GLOBALCONSTANTS DefaultPool_Numeric (* Numeric object pool constants (ID, Scale, Offset, Decimals) *)
  PACKAGE test::FBs::Baumsetzer::Constants;
  VAR_GLOBAL CONSTANT
    InputNumber_Pflanzabstand : logiBUS::utils::conversion::phys::NumericObjectPool_S := (u16ObjId := 9001, r32Scale := 0.001, i32Offset := 0, u8Decimals := 3);
    InputNumber_Luftversatz : logiBUS::utils::conversion::phys::NumericObjectPool_S := (u16ObjId := 9002, r32Scale := 0.1, i32Offset := 0, u8Decimals := 1);
    InputNumber_Wasserversatz : logiBUS::utils::conversion::phys::NumericObjectPool_S := (u16ObjId := 9003, r32Scale := 0.1, i32Offset := 0, u8Decimals := 1);
    InputNumber_Granulatversatz : logiBUS::utils::conversion::phys::NumericObjectPool_S := (u16ObjId := 9004, r32Scale := 0.1, i32Offset := 0, u8Decimals := 1);
    InputNumber_Summer_Dauer : logiBUS::utils::conversion::phys::NumericObjectPool_S := (u16ObjId := 9005, r32Scale := 1.0, i32Offset := 0, u8Decimals := 0);
    InputNumber_Luft_Dauer : logiBUS::utils::conversion::phys::NumericObjectPool_S := (u16ObjId := 9006, r32Scale := 1.0, i32Offset := 0, u8Decimals := 0);
    InputNumber_Wasser_Dauer : logiBUS::utils::conversion::phys::NumericObjectPool_S := (u16ObjId := 9007, r32Scale := 1.0, i32Offset := 0, u8Decimals := 0);
    InputNumber_Granulat_Dauer : logiBUS::utils::conversion::phys::NumericObjectPool_S := (u16ObjId := 9008, r32Scale := 1.0, i32Offset := 0, u8Decimals := 0);
    OutputNumber_12000 : logiBUS::utils::conversion::phys::NumericObjectPool_S := (u16ObjId := 12000, r32Scale := 0.0036, i32Offset := 0, u8Decimals := 1);
    Einsatzstunden : logiBUS::utils::conversion::phys::NumericObjectPool_S := (u16ObjId := 12001, r32Scale := 1.0, i32Offset := 0, u8Decimals := 0);
    Einsatzminuten : logiBUS::utils::conversion::phys::NumericObjectPool_S := (u16ObjId := 12002, r32Scale := 1.0, i32Offset := 0, u8Decimals := 0);
    OutputNumber_Baeume_gepflanzt : logiBUS::utils::conversion::phys::NumericObjectPool_S := (u16ObjId := 12003, r32Scale := 1.0, i32Offset := 0, u8Decimals := 0);
    OutputNumber_12004 : logiBUS::utils::conversion::phys::NumericObjectPool_S := (u16ObjId := 12004, r32Scale := 0.0036, i32Offset := 0, u8Decimals := 1);
    OutputNumber_12005 : logiBUS::utils::conversion::phys::NumericObjectPool_S := (u16ObjId := 12005, r32Scale := 0.0036, i32Offset := 0, u8Decimals := 1);
    OutputNumber_12006 : logiBUS::utils::conversion::phys::NumericObjectPool_S := (u16ObjId := 12006, r32Scale := 0.0036, i32Offset := 0, u8Decimals := 1);
    OutputNumber_12007 : logiBUS::utils::conversion::phys::NumericObjectPool_S := (u16ObjId := 12007, r32Scale := 0.0036, i32Offset := 0, u8Decimals := 1);
  END_VAR
END_GLOBALCONSTANTS
